FUNCTION_BLOCK ReactorActuators (* Composite Function Block Type *)
  (* Standard: 61499-2 *)
  (* Version 0.0, 11/16/2023, SESA371406, Schneider Electric, template *)
  PACKAGE SE.Nereda;
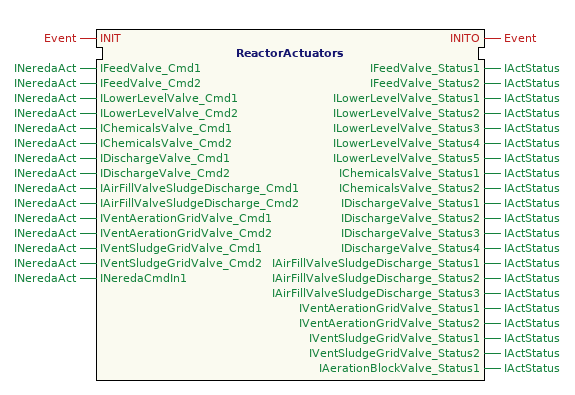
  EVENT_INPUT
    INIT;
  END_EVENT
  EVENT_OUTPUT
    INITO;
  END_EVENT
  SOCKETS
    IFeedValve_Cmd1 : INeredaAct;
    IFeedValve_Cmd2 : INeredaAct;
    ILowerLevelValve_Cmd1 : INeredaAct;
    ILowerLevelValve_Cmd2 : INeredaAct;
    IChemicalsValve_Cmd1 : INeredaAct;
    IChemicalsValve_Cmd2 : INeredaAct;
    IDischargeValve_Cmd1 : INeredaAct;
    IDischargeValve_Cmd2 : INeredaAct;
    IAirFillValveSludgeDischarge_Cmd1 : INeredaAct;
    IAirFillValveSludgeDischarge_Cmd2 : INeredaAct;
    IVentAerationGridValve_Cmd1 : INeredaAct;
    IVentAerationGridValve_Cmd2 : INeredaAct;
    IVentSludgeGridValve_Cmd1 : INeredaAct;
    IVentSludgeGridValve_Cmd2 : INeredaAct;
    INeredaCmdIn1 : INeredaAct;
  END_SOCKETS
  PLUGS
    IFeedValve_Status1 : IActStatus;
    IFeedValve_Status2 : IActStatus;
    ILowerLevelValve_Status1 : IActStatus;
    ILowerLevelValve_Status2 : IActStatus;
    ILowerLevelValve_Status3 : IActStatus;
    ILowerLevelValve_Status4 : IActStatus;
    ILowerLevelValve_Status5 : IActStatus;
    IChemicalsValve_Status1 : IActStatus;
    IChemicalsValve_Status2 : IActStatus;
    IDischargeValve_Status1 : IActStatus;
    IDischargeValve_Status2 : IActStatus;
    IDischargeValve_Status3 : IActStatus;
    IDischargeValve_Status4 : IActStatus;
    IAirFillValveSludgeDischarge_Status1 : IActStatus;
    IAirFillValveSludgeDischarge_Status2 : IActStatus;
    IAirFillValveSludgeDischarge_Status3 : IActStatus;
    IVentAerationGridValve_Status1 : IActStatus;
    IVentAerationGridValve_Status2 : IActStatus;
    IVentSludgeGridValve_Status1 : IActStatus;
    IVentSludgeGridValve_Status2 : IActStatus;
    IAerationBlockValve_Status1 : IActStatus;
  END_PLUGS
  (* 01 - FUNCTIONNAL INPUT INTERFACE *)
  (* 00 - INITIALIZATION *)
  (* 05 - LOGIC *)
  (* 06 - HMI INTERFACE *)
  (* 03 - FIELD INTERFACE *)
  (* 02 - FUNCTIONNAL OUTPUT INTERFACE *)
  (* Actuators Status *)
  (* 04 - CHILDREN *)
  (* 4A - TYPICALS *)
  (* Actuators Command *)
  (* Reset All Actuators *)
  (* Actuators Tags : - Feed valve :                                  AV4x101 - Lower level valve :                        AV4x102 - Discharge valve :                         AV4x103 - Vent aeration grid valve :             AV4x107 - Chemicals valve :                         AV4x108 - Air fill valve sludge discharge :    AV4x171 - Vent sludge grid valve :               AV4x172 *)
  (* Not in the control narrative *)
  FBS
    ResetAllValves : ResetValvesManager;
    FeedValve_AV4x101 : ValveS;
    DischargeValve_AV4x103 : ValveS;
    FeedingValve_Status : MultiActStatus;
    DischargeValve_Status : MultiActStatus;
    FeedingValve_Cmd : MultiNeredaCmd;
    DischargeValve_Cmd : MultiNeredaCmd;
    LowerLevelValve_AV4x102 : ValveS;
    LowerLevelValve_Status : MultiActStatus;
    LowerLevelValve_Cmd : MultiNeredaCmd;
    AirFillValveSludgeDischarge_AV4x171 : ValveS;
    AirFillValveSludgeDischarge_Status : MultiActStatus;
    AirFillValveSludgeDischarge_Cmd : MultiNeredaCmd;
    VentAerationGridValve_AV4x107 : ValveS;
    VentAerationGridValve_Status : MultiActStatus;
    VentAerationGridValve_Cmd : MultiNeredaCmd;
    ChemicalsValve_AV4x108 : ValveS;
    MetalDosingValve_Status : MultiActStatus;
    MetalDosingValve_Cmd : MultiNeredaCmd;
    VentSludgeGridValve_AV4x172 : ValveS;
    VentSludgeGridValve_Status : MultiActStatus;
    VentSludgeGridValve_Cmd : MultiNeredaCmd;
    DischargeValve_Status1 : MultiActStatus;
    LowerLevelValve_Status1 : MultiActStatus;
    AerationBlockValve_AV4x170 : ValveS;
    VentSludgeGridValve_Status1 : MultiActStatus;
    VentSludgeGridValve_Cmd1 : MultiNeredaCmd;
  END_FBS
  EVENT_CONNECTIONS
    INIT TO ResetAllValves.INIT;
    ResetAllValves.INITO TO INITO;
  END_CONNECTIONS
  ADAPTER_CONNECTIONS
    IFeedValve_Cmd1 TO FeedingValve_Cmd.F1CE5E5BC0F88348;
    IFeedValve_Cmd2 TO FeedingValve_Cmd.814FBE7646911966;
    IDischargeValve_Cmd1 TO DischargeValve_Cmd.F1CE5E5BC0F88348;
    IDischargeValve_Cmd2 TO DischargeValve_Cmd.814FBE7646911966;
    FeedingValve_Cmd.30D463C0CF465CCB TO FeedValve_AV4x101.476D0447CF6D114C;
    DischargeValve_Cmd.30D463C0CF465CCB TO DischargeValve_AV4x103.476D0447CF6D114C;
    FeedValve_AV4x101.E9B1CB906EB3FD07 TO FeedingValve_Status.18836B5B646921E0;
    DischargeValve_AV4x103.E9B1CB906EB3FD07 TO DischargeValve_Status.18836B5B646921E0;
    FeedingValve_Status.8244952938F4EC92 TO IFeedValve_Status1;
    FeedingValve_Status.3FD61FA75EE1C84B TO IFeedValve_Status2;
    DischargeValve_Status.8244952938F4EC92 TO IDischargeValve_Status1;
    DischargeValve_Status.3FD61FA75EE1C84B TO IDischargeValve_Status2;
    ResetAllValves.2 TO FeedValve_AV4x101.76FFF418213BE03C;
    ResetAllValves.5 TO DischargeValve_AV4x103.76FFF418213BE03C;
    ResetAllValves.9 TO LowerLevelValve_AV4x102.76FFF418213BE03C;
    LowerLevelValve_Cmd.30D463C0CF465CCB TO LowerLevelValve_AV4x102.476D0447CF6D114C;
    LowerLevelValve_AV4x102.E9B1CB906EB3FD07 TO LowerLevelValve_Status.18836B5B646921E0;
    ILowerLevelValve_Cmd1 TO LowerLevelValve_Cmd.F1CE5E5BC0F88348;
    ILowerLevelValve_Cmd2 TO LowerLevelValve_Cmd.814FBE7646911966;
    LowerLevelValve_Status.8244952938F4EC92 TO ILowerLevelValve_Status1;
    LowerLevelValve_Status.3FD61FA75EE1C84B TO ILowerLevelValve_Status2;
    ResetAllValves.11 TO AirFillValveSludgeDischarge_AV4x171.76FFF418213BE03C;
    AirFillValveSludgeDischarge_AV4x171.E9B1CB906EB3FD07 TO AirFillValveSludgeDischarge_Status.18836B5B646921E0;
    AirFillValveSludgeDischarge_Cmd.30D463C0CF465CCB TO AirFillValveSludgeDischarge_AV4x171.476D0447CF6D114C;
    AirFillValveSludgeDischarge_Status.8244952938F4EC92 TO IAirFillValveSludgeDischarge_Status1;
    AirFillValveSludgeDischarge_Status.3FD61FA75EE1C84B TO IAirFillValveSludgeDischarge_Status2;
    IAirFillValveSludgeDischarge_Cmd1 TO AirFillValveSludgeDischarge_Cmd.F1CE5E5BC0F88348;
    IAirFillValveSludgeDischarge_Cmd2 TO AirFillValveSludgeDischarge_Cmd.814FBE7646911966;
    ResetAllValves.12 TO VentAerationGridValve_AV4x107.76FFF418213BE03C;
    VentAerationGridValve_Cmd.30D463C0CF465CCB TO VentAerationGridValve_AV4x107.476D0447CF6D114C;
    VentAerationGridValve_AV4x107.E9B1CB906EB3FD07 TO VentAerationGridValve_Status.18836B5B646921E0;
    VentAerationGridValve_Status.8244952938F4EC92 TO IVentAerationGridValve_Status1;
    VentAerationGridValve_Status.3FD61FA75EE1C84B TO IVentAerationGridValve_Status2;
    IVentAerationGridValve_Cmd1 TO VentAerationGridValve_Cmd.F1CE5E5BC0F88348;
    IVentAerationGridValve_Cmd2 TO VentAerationGridValve_Cmd.814FBE7646911966;
    ResetAllValves.14 TO ChemicalsValve_AV4x108.76FFF418213BE03C;
    ChemicalsValve_AV4x108.E9B1CB906EB3FD07 TO MetalDosingValve_Status.18836B5B646921E0;
    MetalDosingValve_Cmd.30D463C0CF465CCB TO ChemicalsValve_AV4x108.476D0447CF6D114C;
    IChemicalsValve_Cmd1 TO MetalDosingValve_Cmd.F1CE5E5BC0F88348;
    IChemicalsValve_Cmd2 TO MetalDosingValve_Cmd.814FBE7646911966;
    MetalDosingValve_Status.8244952938F4EC92 TO IChemicalsValve_Status1;
    MetalDosingValve_Status.3FD61FA75EE1C84B TO IChemicalsValve_Status2;
    DischargeValve_Status.3A373E4DF127E388 TO IDischargeValve_Status3;
    DischargeValve_Status.88456893CB21FD74 TO DischargeValve_Status1.18836B5B646921E0;
    AirFillValveSludgeDischarge_Status.3A373E4DF127E388 TO IAirFillValveSludgeDischarge_Status3;
    LowerLevelValve_Status.3A373E4DF127E388 TO ILowerLevelValve_Status3;
    LowerLevelValve_Status.88456893CB21FD74 TO LowerLevelValve_Status1.18836B5B646921E0;
    VentSludgeGridValve_Cmd.30D463C0CF465CCB TO VentSludgeGridValve_AV4x172.476D0447CF6D114C;
    ResetAllValves.15 TO VentSludgeGridValve_AV4x172.76FFF418213BE03C;
    VentSludgeGridValve_AV4x172.E9B1CB906EB3FD07 TO VentSludgeGridValve_Status.18836B5B646921E0;
    IVentSludgeGridValve_Cmd1 TO VentSludgeGridValve_Cmd.F1CE5E5BC0F88348;
    IVentSludgeGridValve_Cmd2 TO VentSludgeGridValve_Cmd.814FBE7646911966;
    VentSludgeGridValve_Status.8244952938F4EC92 TO IVentSludgeGridValve_Status1;
    VentSludgeGridValve_Status.3FD61FA75EE1C84B TO IVentSludgeGridValve_Status2;
    DischargeValve_Status1.3FD61FA75EE1C84B TO IDischargeValve_Status4;
    LowerLevelValve_Status1.8244952938F4EC92 TO ILowerLevelValve_Status4;
    LowerLevelValve_Status1.3FD61FA75EE1C84B TO ILowerLevelValve_Status5;
    VentSludgeGridValve_Cmd1.30D463C0CF465CCB TO AerationBlockValve_AV4x170.476D0447CF6D114C;
    AerationBlockValve_AV4x170.E9B1CB906EB3FD07 TO VentSludgeGridValve_Status1.18836B5B646921E0;
    INeredaCmdIn1 TO VentSludgeGridValve_Cmd1.F1CE5E5BC0F88348;
    VentSludgeGridValve_Status1.8244952938F4EC92 TO IAerationBlockValve_Status1;
  END_CONNECTIONS
END_FUNCTION_BLOCK
